(* CODESYS project cGit-issue1

Project tree, tasks and I/O mapping:
  Device : CODESYS Control Win V3, 3S - Smart Software Solutions GmbH, version 3.5.19.0
    application Application
      libraries: Standard, 3.5.18.0 (System); Util, 3.5.19.0 (System); VisuDialogs, * (System)
      task AlarmManagerTask (cyclic, interval 50 ms, priority 31) calls AlarmManager.Alarm_Prg
      task MainTask (cyclic, interval t#20ms, priority 1) calls PLC_PRG, Simulation
      task VISU_TASK (cyclic, interval 100 ms, priority 31) calls VisuElems.Visu_Prg
      Alarm Configuration
        text list ag01
        alarm group ag01
        alarm class AlarmClass (priority 0, acknowledge ACK)
        AlarmStorage
        alarm class Error (priority 10, acknowledge REP_ACK)
        alarm class Info (priority 100, acknowledge REP)
        alarm class Warning (priority 30, acknowledge REP)
      visualisation Diagnosis
      global variables Glob_Var
      visualisation Live_Visu
      program PLC_PRG [CFC]
      program Signals [LD]
      program Simulation [ST]
      visualisation Visualization
  text list GlobalTextList
*)

// Device/Application/Glob_Var
{attribute 'qualified_only'}
VAR_GLOBAL
//Inputs
	TempActual: REAL:=8.0;
	TempSet: REAL:=8.0;
	DoorOpen: BOOL;
	AlarmThreshold:TIME:=T#10S;
	DoorOpenThreshold:TIME:=T#10S;

//Outputs
	Compressor: BOOL;
	Signal: BOOL;
	Lamp: BOOL;
END_VAR

// Device/Application/PLC_PRG
// The program activates or deactivates the cooling compressor depending on the 
// deviaton of the actual temperature from the septpoint temperature (with a hysteresis)

// TRUE or FALSE of the cooling compresseor is transfered to the signal processing.
PROGRAM PLC_PRG
VAR
	SR_0: SR;
	Hysteresis: REAL:=1.0;
END_VAR

// note: 1 stored wires end on pins the file does not list and are not shown
SR_0(SET1 := Glob_Var.TempActual > Glob_Var.TempSet + Hysteresis, RESET := Glob_Var.TempActual < Glob_Var.TempSet - Hysteresis); // SR
Glob_Var.Compressor := SR_0.Q1;
Signals();

END_PROGRAM

// Device/Application/Signals
PROGRAM Signals
VAR
	TON_0: TON;
	TON_1: TON;
	tSignalTime:TIME:=T#1S;
	BLINK_0: BLINK;
END_VAR

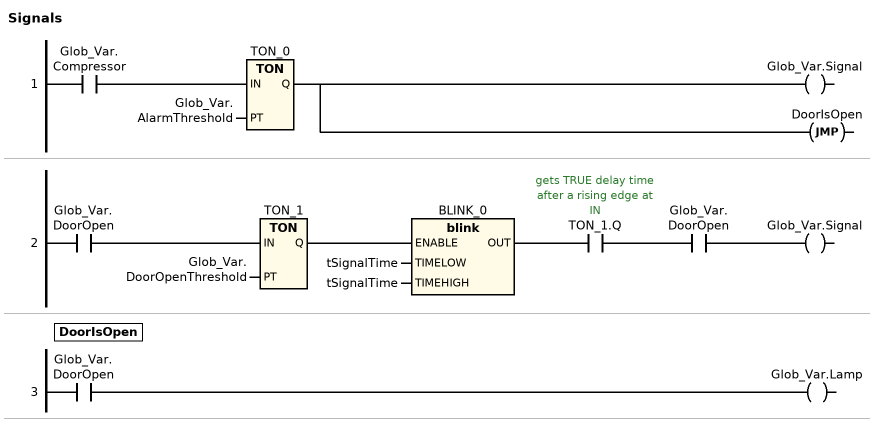
// NETWORK 1
TON_0(IN := Glob_Var.Compressor, PT := Glob_Var.AlarmThreshold); // TON
Glob_Var.Signal := TON_0.Q;
IF TON_0.Q THEN JMP DoorIsOpen; END_IF

// NETWORK 2
//   TON_1.Q: gets TRUE delay time after a rising edge at IN
TON_1(IN := Glob_Var.DoorOpen, PT := Glob_Var.DoorOpenThreshold); // TON
BLINK_0(ENABLE := TON_1.Q, TIMELOW := tSignalTime, TIMEHIGH := tSignalTime); // blink
Glob_Var.Signal := BLINK_0.OUT AND TON_1.Q AND Glob_Var.DoorOpen;

// NETWORK 3
DoorIsOpen:
Glob_Var.Lamp := Glob_Var.DoorOpen;

END_PROGRAM

// Device/Application/Simulation
PROGRAM Simulation
VAR
	T1: TON;					//The temperature is decreased on a time delay, when the comepressor has been activated
	P_Cooling: TIME:=T#500MS;			
	xReduceTemp: BOOL;			//Signal for dereasing the temperature
	T2: TON;					//The temperature is increased on a time delay, when the compressor has been activated 
	P_Environment: TIME:=T#2S;			//Delay time when the door is closed
	P_EnvironmentDoorOpen: TIME:=T#1S;	//Delay time when the door is open
	xRaiseTemp: BOOL;					//Signal for increasing the temperature
	tTemp: TIME;						//Delay time
END_VAR

// After the compressor has been activated due to TempActual being too high, the temperature decreases.
// The temperature is decremented by 0.1°C per cycle after a delay of P_Cooling
IF Glob_Var.Compressor THEN
	T1(IN:= Glob_Var.Compressor, PT:= P_Cooling, Q=>xReduceTemp);
	IF xReduceTemp THEN
		Glob_Var.TempActual := Glob_Var.TempActual-0.1;
		T1(IN:=FALSE);
	END_IF
END_IF

//If the door is open, the warming occurs faster; SEL selects P_EnvironmentDoorOpen
tTemp:=SEL(Glob_Var.DoorOpen, P_Environment, P_EnvironmentDoorOpen);

//If the compressor is not in operation, then the cooling chamber becomes warmer.
//The  temperature is incremented by 0.1°C per cycle after a delay of tTemp
T2(IN:= TRUE, PT:= tTemp, Q=>xRaiseTemp);	
IF xRaiseTemp THEN
	Glob_Var.TempActual := Glob_Var.TempActual + 0.1;
	T2(IN:=FALSE);
END_IF

END_PROGRAM

// Device/Application/Diagnosis
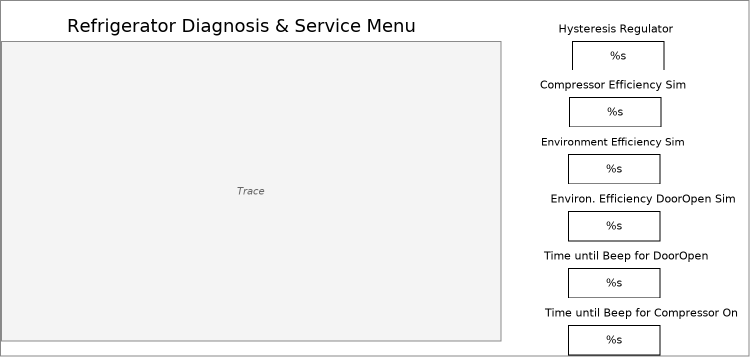
VISUALIZATION Diagnosis  // 750x357
    Trace (1,41 500x300)
    Rectangle (24,11 435x30), "Refrigerator Diagnosis & Service Menu"
    Group (541,14 150x57)
        Rectangle (0,0 150x30), "Hysteresis Regulator"
        Rectangle (31,27 92x30), "%s", text variable: PLC_PRG.Hysteresis
            OnMouseDown: write the text variable via Default
    Group (538,70 150x57)
        Rectangle (0,0 150x30), "Compressor Efficiency Sim"
        Rectangle (31,27 92x30), "%s", text variable: Simulation.P_Cooling
            OnMouseDown: write the text variable via Default
    Group (538,127 150x57)
        Rectangle (0,0 150x30), "Environment Efficiency Sim"
        Rectangle (30,27 92x30), "%s", text variable: Simulation.P_Environment
            OnMouseDown: write the text variable via Default
    Group (538,241 177x57)
        Rectangle (0,0 177x30), "Time until Beep for DoorOpen"
        Rectangle (30,27 92x30), "%s", text variable: Glob_Var.DoorOpenThreshold
            OnMouseDown: write the text variable via Default
    Group (538,298 207x57)
        Rectangle (0,0 207x30), "Time until Beep for Compressor On"
        Rectangle (30,27 92x30), "%s", text variable: Glob_Var.AlarmThreshold
            OnMouseDown: write the text variable via Default
    Rectangle (538,184 210x30), "Environ. Efficiency DoorOpen Sim"
    Rectangle (568,211 92x30), "%s", text variable: Simulation.P_EnvironmentDoorOpen
        OnMouseDown: write the text variable via Default
END_VISUALIZATION

// Device/Application/Live_Visu
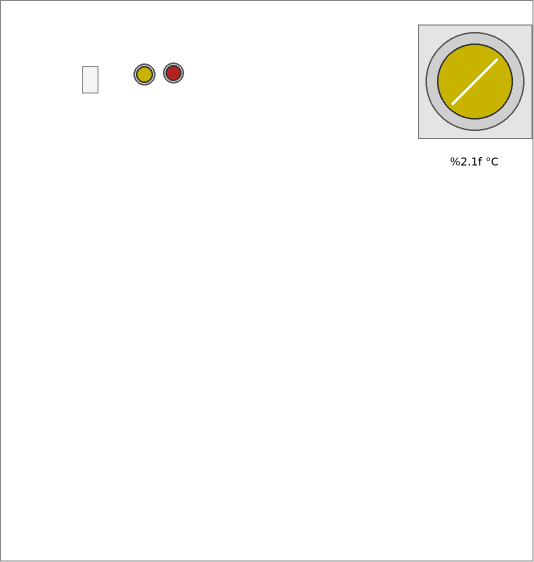
VISUALIZATION Live_Visu  // 534x562
    Polygon (13,14) (261,7) (373,51) (69,61)
    Polygon (77,61) (367,52) (367,75) (76,90)
    Polygon (69,61) (77,61) (77,89) (73,91) (66,89)
    Polygon (13,13) (68,61) (67,91) (13,43)
    Polygon (367,51) (377,51) (376,73) (367,74)
    Potentiometer360 (418,24 114x115), variable: Glob_Var.TempSet, style: Potentiometer-Potentiometer360-Yellow, scale format: %.0f, scale 3..13
        p2431819421: Outside
        p518627256: °C
    Rectangle (426,145 97x34), "%2.1f °C", text variable: Glob_Var.TempActual
    Lamp1 (132,62 25x25), variable: Glob_Var.Compressor, style: Lamp-Lamp1-Yellow
    Lamp1 (161,61 25x24), variable: Glob_Var.Signal, style: Lamp-Lamp1-Red
    Group (66,75 301x465)
        Polygon (3,17) (301,0) (292,422) (5,465) (2,464)
        Group (0,30 33x119)
            Polygon (2,0) (18,1) (22,11) (28,29) (32,46) (33,67) (31,84) (27,97) (22,108) (16,119) (3,117) (15,97) (18,84) (20,70) (20,48) (15,27) (9,14)
            Polygon (3,0) (0,1) (0,5) (3,8) (5,12) (8,16) (10,20) (12,26) (13,31) (16,40) (17,46) (18,54) (18,62) (18,72) (16,80) (14,89) (11,97) (7,106) (2,117) (4,118) (9,107) (13,100) (17,90) (19,80) (21,69) (21,62) (20,48) (17,36) (15,27) (10,14) (7,7)
    Polygon (13,45) (66,92) (69,539) (12,412)
    Group (65,78 299x482), invisible if: NOT Glob_Var.DoorOpen
        Polygon (1,17) (299,0) (290,422) (3,465) (0,464)
        Group (21,0 278x482)
            Polygon (1,34) (278,0) (270,421) (3,482) (0,481)
            Group (1,69 33x119)
                Polygon (2,0) (18,1) (22,11) (28,29) (32,46) (33,67) (31,84) (27,97) (22,108) (16,119) (3,117) (15,97) (18,84) (20,70) (20,48) (15,27) (9,14)
                Polygon (3,0) (0,1) (0,5) (3,8) (5,12) (8,16) (10,20) (12,26) (13,31) (16,40) (17,46) (18,54) (18,62) (18,72) (16,80) (14,89) (11,97) (7,106) (2,117) (4,118) (9,107) (13,100) (17,90) (19,80) (21,69) (21,62) (20,48) (17,36) (15,27) (10,14) (7,7)
    RockerSwitch (82,66 16x27), variable: Glob_Var.DoorOpen, behaviour: TOGGLE, style: Switch-RockerSwitch-Gray
END_VISUALIZATION

// Device/Application/Visualization
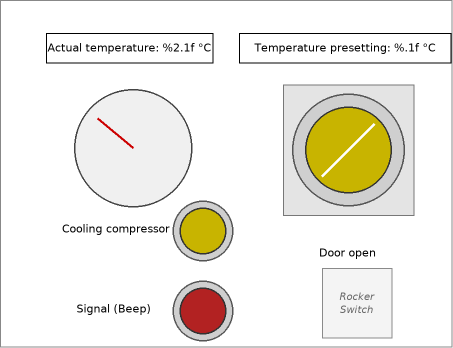
VISUALIZATION Visualization  // 453x348
    Rectangle (46,33 167x30), "Actual temperature: %2.1f °C", text variable: Glob_Var.TempActual
    Lamp1 (168,196 70x70), variable: Glob_Var.Compressor, style: Lamp-Lamp1-Yellow
    Rectangle (239,33 212x30), "Temperature presetting: %.1f °C", text variable: Glob_Var.TempSet
        OnMouseDown: write the text variable via Default, min 3, max 12
    Potentiometer360 (283,84 131x132), variable: Glob_Var.TempSet, style: Potentiometer-Potentiometer360-Yellow, scale format: %.0f, scale 3..13
        p2431819421: Outside
        p518627256: °C
    Meter180 (49,89 168x118), value: Glob_Var.TempActual, style: Meter-Meter180-Gray, scale format: %.1f, scale 0..20
    Rectangle (41,214 150x30), "Cooling compressor"
    Lamp1 (168,276 70x70), variable: Glob_Var.Signal, style: Lamp-Lamp1-Red
    Rectangle (39,294 150x30), "Signal (Beep)"
    RockerSwitch (322,268 70x70), variable: Glob_Var.DoorOpen, behaviour: TOGGLE, style: Switch-RockerSwitch-Gray
    Rectangle (313,238 69x30), "Door open", text variable: Glob_Var.TempSet
END_VISUALIZATION

(* text list ag01 (id | default)
   |  *)
